{attribute 'OPC.UA.DA' := '1'}
FUNCTION_BLOCK Sh10pilShutter EXTENDS ShutterBase
VAR_INPUT
END_VAR
VAR_OUTPUT
END_VAR
VAR
	{attribute 'OPC.UA.DA' := '0'}
	_config : Sh10pilShutterConfig;		
	{attribute 'OPC.UA.DA' := '0'}
	IoSh10pilShutter : IoSh10pilShutter;
	
	{attribute 'OPC.UA.DA' := '0'}
	_deliverMessages : INT;
	
	ShutterIrisPositionMsg : STRING(255);
	
	{region 'Commands'}
	
	{attribute 'OPC.UA.DA' := '0'}
	_open : BOOL;
	{attribute 'OPC.UA.DA' := '0'}
	_close : BOOL;
	{attribute 'OPC.UA.DA' := '0'}			  		   
	_raiseProperties : BOOL;
			
	{endregion}		

	{attribute 'OPC.UA.DA' := '0'}
	_initDevice : BOOL;	
	
	{attribute 'OPC.UA.DA' := '0'}
	_itemScheduler : INT;	
	{attribute 'OPC.UA.DA' := '0'}
	_itemOpen : INT;
	{attribute 'OPC.UA.DA' := '0'}
	_itemClose : INT;
	{attribute 'OPC.UA.DA' := '0'}
	_pulseGenerator : TON;	
	{attribute 'OPC.UA.DA' := '0'}
	_pulseOpen : TON;
	{attribute 'OPC.UA.DA' := '0'}
	_pulseClose : TON;
	{attribute 'OPC.UA.DA' := '0'}
	_pulseTimeout : TON;		
	{attribute 'OPC.UA.DA' := '0'}
	_itemRaisedProperties : INT;	
	
	{attribute 'OPC.UA.DA' := '0'}
	message : STRING;
	
END_VAR

// Init device
InitDevice();

CASE _deliverMessages OF			
	EFeedbackMsgSh10pil.ShutterIrisPositionMsg :	
		ShutterIrisPositionMsg := message;	
END_CASE
		
// Commands		
ManualOpen(_open);
ManualClose(_close);
RaisePropertiesChanged(_raiseProperties);

IF (NOT _open AND NOT _close AND NOT _raiseProperties) THEN
	_deliverMessages := 0;
	MessageScheduler();
END_IF

METHOD FB_init : BOOL
VAR_INPUT
	bInitRetains : BOOL; // if TRUE, the retain variables are initialized (warm start / cold start)
	bInCopyCode : BOOL;  // if TRUE, the instance afterwards gets moved into the copy code (online change)
	Config : Sh10pilShutterConfig;
END_VAR
IF Config.IsEnabled THEN
	_config := Config;
	
	SUPER^._shutterConfig.Name := Config.Name;
	SUPER^._shutterConfig.DeviceID := Config.DeviceID;
	SUPER^._shutterConfig.IsEnabled := Config.IsEnabled;
	SUPER^._shutterConfig.LogLevel := Config.LogLevel;
	
	SUPER^.Name := Config.Name;
	SUPER^.DeviceID := Config.DeviceID;	
	THIS^.Family := DeviceFamily.Shutter;
		
	_Logger.Information(_message.Reset().Append('Init ').
							Append('{').Append(TO_STRING(THIS^.Family)).Append('} - ').
							Append('{').Append(TO_STRING(Config.Name)).Append('}').ToString());																													
END_IF
END_METHOD

METHOD InitDevice
VAR_INPUT
END_VAR
IF NOT _initDevice THEN	
	_logger.Information(_message.Reset().
								Append(_config.Name).
								Append(' - Init device').ToString());
	
	THIS^.SetDone();
	_initDevice := TRUE;	
END_IF
END_METHOD

{attribute 'TcRpcEnable' := '1'}
METHOD PROTECTED ManualClose
VAR_INPUT
	Execute : BOOL;
END_VAR
IF Execute THEN	
	_close := TRUE;
	
	CASE _itemClose OF
		0: _logger.Information(_message.Reset().
							Append(_config.Name).
							Append(' - Close').ToString());
							
			_itemClose := 1;
							
		1: //Wait until the shutter is opened 
			IF IoSh10pilShutter.InputMagneticSwitch1 AND NOT IoSh10pilShutter.InputMagneticSwitch2 THEN
				_itemClose := 2;
			ELSE 
				// Raised timer 
				IF _pulseTimeout.Q THEN
					_pulseTimeout(IN := FALSE);
					
					_itemClose := 2;
				ELSE
					_pulseTimeout(IN := TRUE, PT := T#100MS);	
				END_IF	
			END_IF 
			
		2: IF _pulseOpen.Q THEN
				_pulseOpen(IN := FALSE);
				
				IoSh10pilShutter.OutputSwitchContactClosure := FALSE;
				_close := FALSE;
				_itemClose := 0;
			ELSE
				_pulseOpen(IN := TRUE, PT := T#10MS);	
			END_IF		
							
	END_CASE

END_IF
END_METHOD

{attribute 'TcRpcEnable' := '1'}
METHOD PROTECTED ManualOpen
VAR_INPUT
	Execute : BOOL;
END_VAR
IF Execute THEN
	_open := TRUE;
	
	CASE _itemOpen OF
		0: _logger.Information(_message.Reset().
							Append(_config.Name).
							Append(' - Open').ToString());
							
			_itemOpen := 1;
							
		1: //Wait until the shutter is closed 
			IF NOT IoSh10pilShutter.InputMagneticSwitch1 AND IoSh10pilShutter.InputMagneticSwitch2 THEN
				_itemOpen := 2;
			ELSE
				// Raised timer 
				IF _pulseTimeout.Q THEN
					_pulseTimeout(IN := FALSE);
					
					_itemOpen := 2;
				ELSE
					_pulseTimeout(IN := TRUE, PT := T#100MS);	
				END_IF	
			END_IF 
			
		2: IF _pulseOpen.Q THEN
				_pulseOpen(IN := FALSE);
				
				IoSh10pilShutter.OutputSwitchContactClosure := TRUE;
				_open := FALSE;
				_itemOpen := 0;
			ELSE
				_pulseOpen(IN := TRUE, PT := T#400MS);	
			END_IF		
							
	END_CASE
	
END_IF
END_METHOD

METHOD MessageScheduler
VAR_INPUT
END_VAR
IF _pulseGenerator.Q THEN
	_pulseGenerator(IN := FALSE, PT := T#10MS);
	
	ShutterIrisPosition();
ELSE
	_pulseGenerator(IN := TRUE, PT := T#100MS);		
END_IF
END_METHOD

{attribute 'TcRpcEnable' := '1'}
METHOD RaisePropertiesChanged
VAR_INPUT
	Execute : BOOL;
END_VAR
IF Execute THEN		
	_raiseProperties := TRUE;	
	
	IF _pulseGenerator.Q THEN
		_pulseGenerator(IN := FALSE, PT := T#10MS);
		
		CASE _itemRaisedProperties OF		
			0: ShutterIrisPositionMsg := ' ';
				_itemRaisedProperties := 1;
			
			1: ShutterIrisPosition();		   
				_itemRaisedProperties := 10;
				
			10: 
				_logger.Information(_message.Reset().
								    Append(_config.Name).
								    Append(' - RaisePropertiesChanged').ToString());
				_raiseProperties := FALSE;
				_itemRaisedProperties := 0;
		
		END_CASE
	
	ELSE
		_pulseGenerator(IN := TRUE, PT := T#200MS);	
	END_IF
		
END_IF
END_METHOD

METHOD ShutterIrisPosition 
VAR_INPUT
END_VAR
VAR 
	close : STRING := 'CLOSE';
	open : STRING := 'OPEN';
	error : STRING := 'ERROR';
END_VAR
_deliverMessages := EFeedbackMsgEd12dss.ShutterIrisPositionMsg;

IF IoSh10pilShutter.InputMagneticSwitch1 AND NOT IoSh10pilShutter.InputMagneticSwitch2 THEN
	message := open; 		
ELSIF NOT IoSh10pilShutter.InputMagneticSwitch1 AND IoSh10pilShutter.InputMagneticSwitch2 THEN
	message := close; 
ELSIF IoSh10pilShutter.InputMagneticSwitch1 AND IoSh10pilShutter.InputMagneticSwitch2 THEN
	message := error; 
END_IF
END_METHOD

END_FUNCTION_BLOCK

(* stored: Version 1.1.0.1, ProductVersion 3.1.4024.12
   POU Sh10pilShutter: Id {38ecd2b8-a49e-4667-b446-b434800fc359}, SpecialFunc None
   Folder Commands: Id {784605ba-45c7-45f0-a28b-57422efcb1aa}
   Method FB_init: Id {14423b6a-7575-4fca-aa98-5094170539ad}
   Method InitDevice: Id {8a864f3b-4dae-414c-8cfe-8cb22c59f992}
   Method ManualClose: Id {d64b9230-4ec8-4e0e-be01-d7c4a304df93}
   Method ManualOpen: Id {1066cd26-cc42-48ca-96ef-2f5008eb325c}
   Method MessageScheduler: Id {b6a4bfb0-e437-4676-9ba5-04c6dc6ed13f}
   Method RaisePropertiesChanged: Id {12cf85a0-0b5e-4c9f-96ad-d065b959afd8}
   Method ShutterIrisPosition: Id {f9d6e180-b842-4b68-9a95-e17a0d6fef6f} *)
